FUNCTION_BLOCK FB01
VAR_INPUT
	input1: BOOL;
END_VAR
VAR_OUTPUT
	output1: bool;
END_VAR
VAR
END_VAR

output1:=input1;

END_FUNCTION_BLOCK

(* stored: Version 1.1.0.1, ProductVersion 3.1.4024.11
   POU FB01: Id {74de3924-ae28-4c51-8ac2-79a2615fb79c}, SpecialFunc None *)
